// TIA Portal V17 export
// export: Created 2024-06-16T17:47:31.0498791Z, ExportSetting WithDefaults, DisplayName Totally Integrated Automation Portal, DisplayVersion V17, DisplayName TIA Portal Openness, DisplayVersion V17, DisplayName TIA Portal Version Control Interface, DisplayVersion V17, DisplayName STEP 7 Professional, DisplayVersion V17, DisplayName STEP 7 Safety, DisplayVersion V17, DisplayName WinCC Professional, DisplayVersion V17
DATA_BLOCK "St3_In"   // DB305
{ S7_Optimized_Access := 'TRUE' }
VERSION : 0.1
// stored: AutoNumber false, DBAccessibleFromOPCUA true, DBAccessibleFromWebserver true, IsOnlyStoredInLoadMemory false, IsRetainMemResEnabled false, IsWriteProtectedInAS false, MemoryReserve 100
   VAR
      TrappeEntree_Ouvert : Bool;   // Trappe d'entrée : Ouverte
      TrappeEntree_Fermee : Bool;   // Trappe d'entrée : Fermée
      TrappeSortie_Ouvert : Bool;   // Trappe de sortie : Ouverte
      TrappeSortie_Fermee : Bool;   // Trappe de sortie : Fermée
      Obturateur_Ouvert : Bool;   // Obturateur : Ouvert
      Obturateur_Fermee : Bool;   // Obturateur : Fermé
      PorteRX_Ouvert : Bool;   // Porte RX : Ouverte (Homme)
      PorteRX_Fermee : Bool;   // Porte RX : Ferméee (Homme)
      Cpt_RX1 : Bool;   // Présence barquette en début de RX : RX1
      Cpt_RX2 : Bool;   // Détection butée à came : RX2
      Cpt_RX3 : Bool;   // Détection butée pivot : RX3
      Vy_Orange : Bool;   // Obturateur Fermée + RX Actif
      Vy_Rouge : Bool;   // Obturateur Ouvert + RX Actif
   END_VAR
BEGIN
END_DATA_BLOCK
